// TIA Portal project "Diag_checking" (V17)

(* hardware
DEVICE "ET-200SP"  ET 200SP-Station
   slot 0: "Rack_0"  Rack  6ES5 710-8MAx1
   slot 1: "TEST_ET200SP"  CPU 1510SP-1 PN  6ES7 510-1DJ01-0AB0  V2.9
      slot 32768: "PROFINET interface_1"  X1
   slot 2: "Server module_1"  Server module  6ES7 193-6PA00-0AA0  V1.1
      slot 1: "Server module_1"  Server module
   slot 127: "BA 2xRJ45"  BA 2xRJ45  6ES7 193-6AR00-0AA0  V0.0
      slot 32769: "Port_1"  X1 P1  6ES7 193-6AR00-0AA0
      slot 32770: "Port_2"  X1 P2  6ES7 193-6AR00-0AA0
DEVICE "S7-1200"  S7-1200 Station
   slot 0: "Rack_0"  S7-1200 Rack  Rack  V1.0
   slot 1: "TEST_S7-1200"  CPU 1212C AC/DC/Rly  6ES7 212-1BE40-0XB0  V4.5
   slot 2: "AI 4xTC_1"  6ES7 231-5QD30-0XB0  V1.0
   slot 3: "AI 4x13BIT_1"  6ES7 231-4HD32-0XB0  V2.1
*)

// ===== PLC "TEST_ET200SP"  CPU 1510SP-1 PN =====

ORGANIZATION_BLOCK "Main"   // OB1, LAD, ProgramCycle
TITLE = "Main Program Sweep (Cycle)"
{ S7_Optimized_Access := 'TRUE' }
VERSION : 0.1
   VAR_INPUT
      Initial_Call : Bool;   // Initial call of this OB
      Remanence : Bool;   // =True, if remanent data are available
   END_VAR
BEGIN
END_ORGANIZATION_BLOCK

// ===== PLC "TEST_S7-1200"  CPU 1212C AC/DC/Rly =====

VAR_GLOBAL   // PLC tag table "Default tag table"
   "Clock_Byte" AT %MB0 : Byte;
   "Clock_10Hz" AT %M0.0 : Bool;
   "Clock_5Hz" AT %M0.1 : Bool;
   "Clock_2.5Hz" AT %M0.2 : Bool;
   "Clock_2Hz" AT %M0.3 : Bool;
   "Clock_1.25Hz" AT %M0.4 : Bool;
   "Clock_1Hz" AT %M0.5 : Bool;
   "Clock_0.625Hz" AT %M0.6 : Bool;
   "Clock_0.5Hz" AT %M0.7 : Bool;
   "System_Byte" AT %MB1 : Byte;
   "FirstScan" AT %M1.0 : Bool;
   "DiagStatusUpdate" AT %M1.1 : Bool;
   "AlwaysTRUE" AT %M1.2 : Bool;
   "AlwaysFALSE" AT %M1.3 : Bool;
   "Tag_1" AT %M10.0 : Bool;
   "Tag_2" AT %MW0 : Int;
   "Tag_3" AT %MW20 : Int;
END_VAR

// folder: Diagnostics

TYPE "TModuleState"
   STRUCT
      Laddr : Hw_Device;   // Номер hardware ЦПУ / Периферии
      Mode : UInt;   // Режим: 1 - сконфиг. 2 - неисправен. 3 - отключен. 4 - доступен. 5 - есть ошибка(и)
      RetVal : Int;   // Код ошибки: 0 - ошибок нет
      State : Array[0..15] of Bool;   // Состояние
   END_STRUCT;
   // // State[0] : Групповой бит
   // // State[1] : Модуль 0 (slot 0 )
   // // State[2] : Модуль 1 (slot 1) ЦПУ/Периферия
   // // State[3] : Модуль 2 (slot 2)
   // // State[4] : Модуль 3 (slot 3)
   // // State[5] : Модуль 4 (slot 4)
   // // State[6] : Модуль 5 (slot 5)
   // // State[7] : Модуль 6 (slot 6)
   // // State[8] : Модуль 7 (slot 7)
   // // State[9] : Модуль 8 (slot 8)
   // // State[10] : Модуль 9 (slot 9)
   // // State[11] : Модуль 10 (slot 10)
   // // State[12] : Модуль 11 (slot 11)
   // // State[13] : Модуль 12 (slot 12)
   // // State[14] : Модуль 13 (slot 13)
   // // State[15] : Модуль 14 (slot 14)
END_TYPE

TYPE "TDeviceState"
   STRUCT
      Laddr : Hw_IoSystem;   // Номер hardware profinet IO сети
      Mode : UInt;   // Режим: 1 - сконфиг. 2 - неисправен. 3 - отключен. 4 - доступен. 5 - есть ошибка(и)
      RetVal : Int;   // Код ошибки: 0 - ошибок нет
      State : Array[0..63] of Bool;   // Состояние
   END_STRUCT;
   // // State[0] : Групповой бит
   // // State[1] : Устройство 1 (device number 1)
   // // State[2] : Устройство 2 (device number 2)
   // // State[3] : Устройство 3 (device number 3)
   // // State[4] : Устройство 4 (device number 4)
   // // State[5] : Устройство 5 (device number 5)
   // // State[6] : Устройство 6 (device number 6)
   // // State[7] : Устройство 7 (device number 7)
   // // State[8] : Устройство 8 (device number 8)
   // // State[9] : Устройство 9 (device number 9)
   // // State[10] : Устройство 10 (device number 10)
   // // State[11] : Устройство 11 (device number 11)
   // // State[12] : Устройство 12 (device number 12)
   // // State[13] : Устройство 13 (device number 13)
   // // State[14] : Устройство 14 (device number 14)
   // // State[15] : Устройство 15 (device number 15)
   // // State[16] : Устройство 16 (device number 16)
   // // State[17] : Устройство 17 (device number 17)
   // // State[18] : Устройство 18 (device number 18)
   // // State[19] : Устройство 19 (device number 19)
   // // State[20] : Устройство 20 (device number 20)
   // // State[21] : Устройство 21 (device number 21)
   // // State[22] : Устройство 22 (device number 22)
   // // State[23] : Устройство 23 (device number 23)
   // // State[24] : Устройство 24 (device number 24)
   // // State[25] : Устройство 25 (device number 25)
   // // State[26] : Устройство 26 (device number 26)
   // // State[27] : Устройство 27 (device number 27)
   // // State[28] : Устройство 28 (device number 28)
   // // State[29] : Устройство 29 (device number 29)
   // // State[30] : Устройство 30 (device number 30)
   // // State[31] : Устройство 31 (device number 31)
   // // State[32] : Устройство 32 (device number 32)
   // // State[33] : Устройство 33 (device number 33)
   // // State[34] : Устройство 34 (device number 34)
   // // State[35] : Устройство 35 (device number 35)
   // // State[36] : Устройство 36 (device number 36)
   // // State[37] : Устройство 37 (device number 37)
   // // State[38] : Устройство 38 (device number 38)
   // // State[39] : Устройство 39 (device number 39)
   // // State[40] : Устройство 40 (device number 40)
   // // State[41] : Устройство 41 (device number 41)
   // // State[42] : Устройство 42 (device number 42)
   // // State[43] : Устройство 43 (device number 43)
   // // State[44] : Устройство 44 (device number 44)
   // // State[45] : Устройство 45 (device number 45)
   // // State[46] : Устройство 46 (device number 46)
   // // State[47] : Устройство 47 (device number 47)
   // // State[48] : Устройство 48 (device number 48)
   // // State[49] : Устройство 49 (device number 49)
   // // State[50] : Устройство 50 (device number 50)
   // // State[51] : Устройство 51 (device number 51)
   // // State[52] : Устройство 52 (device number 52)
   // // State[53] : Устройство 53 (device number 53)
   // // State[54] : Устройство 54 (device number 54)
   // // State[55] : Устройство 55 (device number 55)
   // // State[56] : Устройство 56 (device number 56)
   // // State[57] : Устройство 57 (device number 57)
   // // State[58] : Устройство 58 (device number 58)
   // // State[59] : Устройство 59 (device number 59)
   // // State[60] : Устройство 60 (device number 60)
   // // State[61] : Устройство 61 (device number 61)
   // // State[62] : Устройство 62 (device number 62)
   // // State[63] : Устройство 63 (device number 63)
END_TYPE

// folder: (top level)

DATA_BLOCK "NETDB"   // DB1
{ S7_Optimized_Access := 'TRUE' }
VERSION : 0.1
   VAR
      dsProfinet : Array[0..4] of "TDeviceState";
      msS71200 : Array[0..4] of "TModuleState";
      msET200SP : Array[0..4] of "TModuleState";
   END_VAR
BEGIN
END_DATA_BLOCK

FUNCTION "Diag" : Void   // FC1, SCL
{ S7_Optimized_Access := 'TRUE' }
VERSION : 0.1
   VAR_TEMP
      i : Int;
   END_VAR
BEGIN

   FOR #i := 0 TO 4 DO
       "NETDB".dsProfinet[#i].Laddr := "Local~PROFINET_IO-System";
       "NETDB".dsProfinet[#i].Mode := INT_TO_UINT(#i + 1);
       "NETDB".dsProfinet[#i].RetVal := DeviceStates(LADDR := "NETDB".dsProfinet[#i].Laddr,
                                                     MODE := "NETDB".dsProfinet[#i].Mode,
                                                     STATE := "NETDB".dsProfinet[#i].State);
   END_FOR;

   FOR #i := 0 TO 4 DO
       "NETDB".msS71200[#i].Laddr := "Local~Device";
       "NETDB".msS71200[#i].Mode := INT_TO_UINT(#i + 1);
       "NETDB".msS71200[#i].RetVal := ModuleStates(LADDR := "NETDB".msS71200[#i].Laddr,
                                                   MODE := "NETDB".msS71200[#i].Mode,
                                                   STATE := "NETDB".msS71200[#i].State);
   END_FOR;

   FOR #i := 0 TO 4 DO
       "NETDB".msET200SP[#i].Laddr := "TEST_ET200SP~PROFINET_interface_1~IODevice";
       "NETDB".msET200SP[#i].Mode := INT_TO_UINT(#i + 1);
       "NETDB".msET200SP[#i].RetVal := ModuleStates(LADDR := "NETDB".msET200SP[#i].Laddr,
                                                    MODE := "NETDB".msET200SP[#i].Mode,
                                                    STATE := "NETDB".msET200SP[#i].State);
   END_FOR;
END_FUNCTION

ORGANIZATION_BLOCK "Main"   // OB1, LAD, ProgramCycle
TITLE = "Main Program Sweep (Cycle)"
{ S7_Optimized_Access := 'TRUE' }
VERSION : 0.1
   VAR_INPUT
      Initial_Call : Bool;   // Initial call of this OB
      Remanence : Bool;   // =True, if remanent data are available
   END_VAR
   VAR_TEMP   // added for the SCL form of the ladder/FBD networks
      _w1 : Bool;
   END_VAR
BEGIN

REGION Network 1
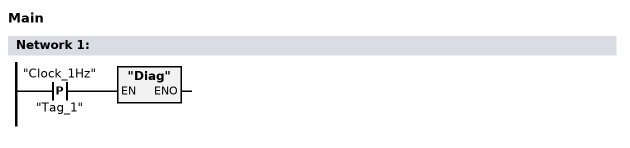
   RUNG wire#powerrail
      P_Contact(operand := "Clock_1Hz", bit := "Tag_1")
      "Diag"()
   END_RUNG
   // the same network as SCL:
   #_w1 := "Clock_1Hz" AND NOT "Tag_1";   // rising edge of "Clock_1Hz"
   "Tag_1" := "Clock_1Hz";
   IF #_w1 THEN "Diag"(); END_IF;
END_REGION
END_ORGANIZATION_BLOCK